Omron CX-Programmer project NuevoProyecto (CX-Programmer 9.31)

# PLC NuevoPLC1: CJ1M CPU11

## Global symbols (name address type ; comment)
C2_FI_CICLE 3101.00 BOOL
C2_MAGATZEM_1_3 3100.00 BOOL
C2_MAGATZEM_2_4 3100.01 BOOL

## Program Cinta2 (cyclic task 0)
Local symbols
AUTO W0.00 BOOL  ; Marca Estat Automatic
BIT_VALIDACIO_SCADA_DESDE_C1 3100.04 BOOL  ; Validació de la emergencia desde el Scada
C2_BE 0.02 BOOL  ; Bolet de Emergència
C2_DM_1_3 0.09 BOOL  ; Detector Magatzem 1-3
C2_DM_2_4 0.11 BOOL  ; Detector Magatzem 2-4
C2_DPC 0.10 BOOL  ; Detector Centre Cinta
C2_EA_0 W130.00 BOOL  ; Etapa Automatic 0
C2_EA_1 W130.01 BOOL  ; Etapa Automatic 1
C2_EA_10 W130.02 BOOL  ; Etapa Automatic 10
C2_EA_11 W130.04 BOOL  ; Etapa Automatic 11
C2_EA_12 W130.05 BOOL  ; Etapa Automatic 12
C2_EA_20 W130.03 BOOL  ; Etapa Automatic 20
C2_EA_21 W130.06 BOOL  ; Etapa Automatic 21
C2_EA_22 W130.07 BOOL  ; Etapa Automatic 22
C2_EA_30 W130.08 BOOL  ; Etapa Automatic 30
C2_EA_31 W130.09 BOOL  ; Etapa Automatic 31
C2_EM_0 W120.00 BOOL  ; Etapa Manual 0
C2_EM_1 W120.01 BOOL  ; Etapa Manual 1
C2_EM_2 W120.02 BOOL  ; Etapa Manual 2
C2_EM_3 W120.03 BOOL  ; Etapa Manual 3
C2_E_A1 W100.00 BOOL
C2_E_A2 W100.03 BOOL
C2_E_D1 W100.06 BOOL
C2_E_D2 W100.07 BOOL
C2_E_F1 W100.01 BOOL
C2_E_F4 W100.04 BOOL
C2_E_F41 W100.05 BOOL
C2_HEMER 1.07 BOOL  ; Pilot Emergència
C2_HMA 1.05 BOOL  ; Pilot mode automàtic
C2_HMM 1.06 BOOL  ; Pilot mode manual
C2_JOYSTICK_FWD 0.03 BOOL  ; Joystick Forward
C2_JOYSTICK_RWD 0.04 BOOL  ; Joystick Reward
C2_MOTOR_FWD 1.09 BOOL  ; Avançament de la cinta
C2_MOTOR_RWD 1.10 BOOL  ; Retrocés de la cinta
C2_PILOT_MARXA 1.00 BOOL  ; Pilot cinta marxa
C2_PM 0.00 BOOL  ; Polsador de Marxa
C2_PP 0.01 BOOL  ; Polsador de Aturada
C2_P_Rearme 0.05 BOOL  ; Polsador de Rearmament
C2_SCADA_JOYSTICK_FWD W101.10 BOOL  ; Joystick SCADA Forward
C2_SCADA_JOYSTICK_RWD W101.11 BOOL  ; Joystick SCADA  Reward
C2_SMA 0.06 BOOL  ; Selector Manual Automatic
CINTA1_REARMADA W300.00 BOOL
COMANDES_SENSE_FINALITZAR 3100.10 BOOL
CT1_MAGATZEM1_3 3100.00 BOOL  ; Ordre peça Magatzem 1-3
CT1_MAGATZEM2_4 3100.01 BOOL  ; Ordre peça Magatzem 2-4
CT2_EMER_LOG 3101.02 BOOL
CT2_FI_CICLE_COM 3101.00 BOOL  ; Ordre de CT2 a CT1, cicle finalitzat
CT2_P_EMER_FIS 3101.03 BOOL
EMER_DESDE_C1 3100.08 BOOL
FI_DE_TOTES_COMADES 3100.09 BOOL
MAN W0.01 BOOL  ; Marca Estat Manual
MEM_FI_COMANDES W100.02 BOOL
M_First_Scan W500.00 BOOL  ; Marca de First Scan
REARMAMENT_C2 W300.10 BOOL
REAR_C1 3100.07 BOOL
REAR_C2 3101.06 BOOL
REAR_CINTES W500.01 BOOL  ; Cinta 1 i Cinta 2 rearmades
RESET_FI_CICLE 3100.05 BOOL
SENYAL_PEÇA_DEIXADA 0.12 BOOL
VAL_TEMPORAL_SCADA W0.08 BOOL

### Section INICIALITZACIÓ_I_ETAPA_ACTIVA_GEMMA

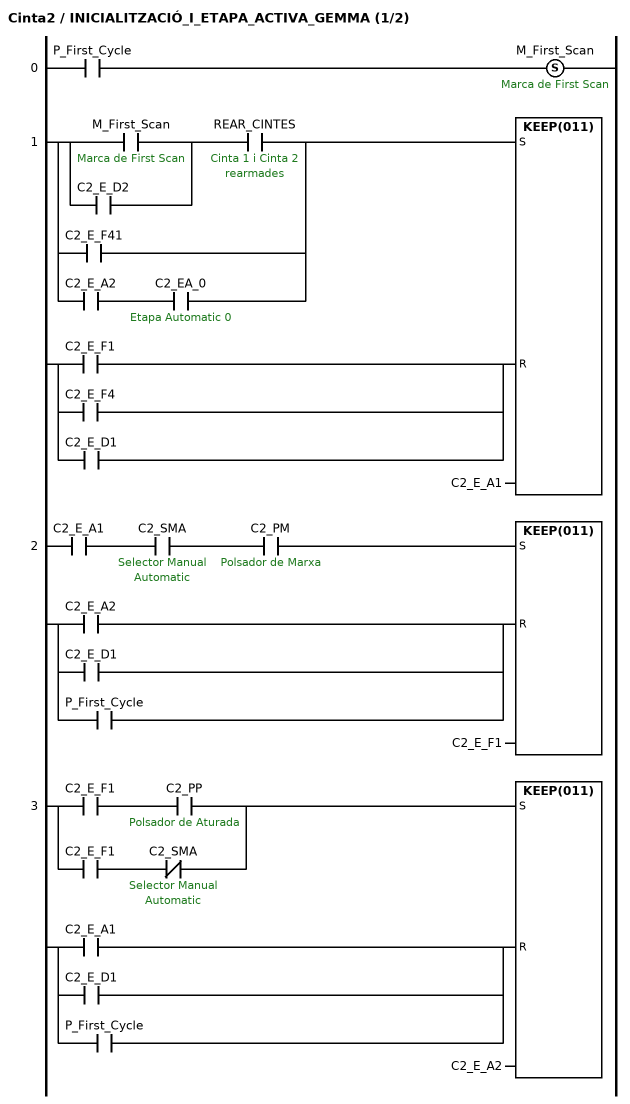
; rung 0
LD P_First_Cycle
SET M_First_Scan  ; Marca de First Scan
; rung 1
LD M_First_Scan  ; Marca de First Scan
OR C2_E_D2
AND REAR_CINTES  ; Cinta 1 i Cinta 2 rearmades
OR C2_E_F41
LD C2_E_A2
AND C2_EA_0  ; Etapa Automatic 0
ORLD
LD C2_E_F1
OR C2_E_F4
OR C2_E_D1
KEEP(011) C2_E_A1
; rung 2
LD C2_E_A1
AND C2_SMA  ; Selector Manual Automatic
AND C2_PM  ; Polsador de Marxa
LD C2_E_A2
OR C2_E_D1
OR P_First_Cycle
KEEP(011) C2_E_F1
; rung 3
LD C2_E_F1
AND C2_PP  ; Polsador de Aturada
LD C2_E_F1
ANDNOT C2_SMA  ; Selector Manual Automatic
ORLD
LD C2_E_A1
OR C2_E_D1
OR P_First_Cycle
KEEP(011) C2_E_A2

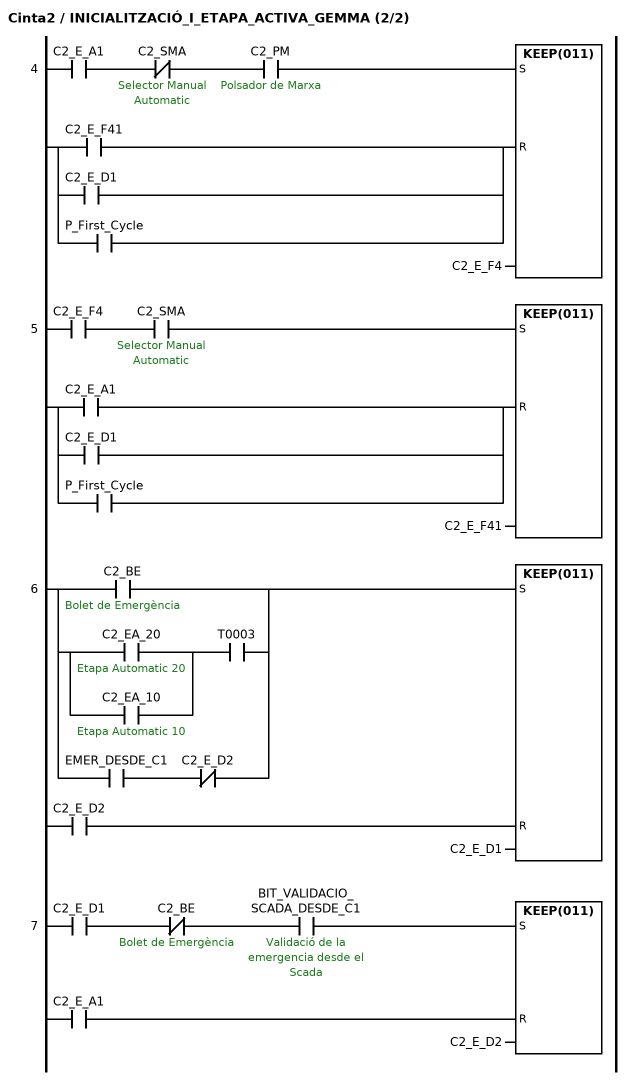
; rung 4
LD C2_E_A1
ANDNOT C2_SMA  ; Selector Manual Automatic
AND C2_PM  ; Polsador de Marxa
LD C2_E_F41
OR C2_E_D1
OR P_First_Cycle
KEEP(011) C2_E_F4
; rung 5
LD C2_E_F4
AND C2_SMA  ; Selector Manual Automatic
LD C2_E_A1
OR C2_E_D1
OR P_First_Cycle
KEEP(011) C2_E_F41
; rung 6
LD C2_BE  ; Bolet de Emergència
LD C2_EA_20  ; Etapa Automatic 20
OR C2_EA_10  ; Etapa Automatic 10
AND T0003
ORLD
LD EMER_DESDE_C1
ANDNOT C2_E_D2
ORLD
LD C2_E_D2
KEEP(011) C2_E_D1
; rung 7
LD C2_E_D1
ANDNOT C2_BE  ; Bolet de Emergència
AND BIT_VALIDACIO_SCADA_DESDE_C1  ; Validació de la emergencia desde el Scada
LD C2_E_A1
KEEP(011) C2_E_D2

### Section ACCIONS_GEMMA

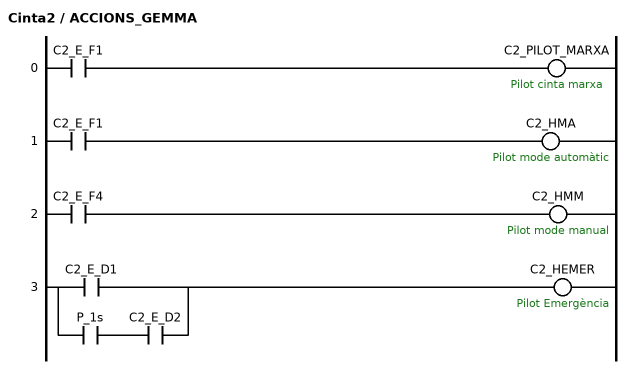
; rung 0
LD C2_E_F1
OUT C2_PILOT_MARXA  ; Pilot cinta marxa
; rung 1
LD C2_E_F1
OUT C2_HMA  ; Pilot mode automàtic
; rung 2
LD C2_E_F4
OUT C2_HMM  ; Pilot mode manual
; rung 3
LD C2_E_D1
LD P_1s
AND C2_E_D2
ORLD
OUT C2_HEMER  ; Pilot Emergència

### Section E_F1

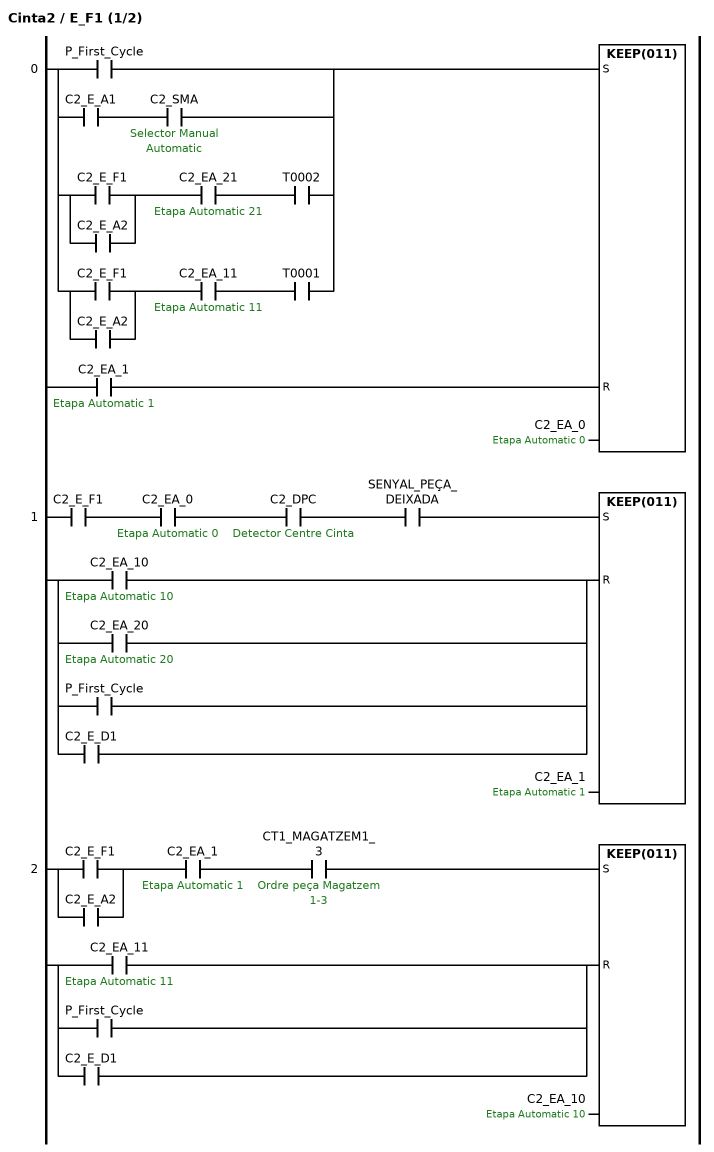
; rung 0
LD P_First_Cycle
LD C2_E_A1
AND C2_SMA  ; Selector Manual Automatic
ORLD
LD C2_E_F1
OR C2_E_A2
AND C2_EA_21  ; Etapa Automatic 21
AND T0002
ORLD
LD C2_E_F1
OR C2_E_A2
AND C2_EA_11  ; Etapa Automatic 11
AND T0001
ORLD
LD C2_EA_1  ; Etapa Automatic 1
KEEP(011) C2_EA_0  ; Etapa Automatic 0
; rung 1
LD C2_E_F1
AND C2_EA_0  ; Etapa Automatic 0
AND C2_DPC  ; Detector Centre Cinta
AND SENYAL_PEÇA_DEIXADA
LD C2_EA_10  ; Etapa Automatic 10
OR C2_EA_20  ; Etapa Automatic 20
OR P_First_Cycle
OR C2_E_D1
KEEP(011) C2_EA_1  ; Etapa Automatic 1
; rung 2
LD C2_E_F1
OR C2_E_A2
AND C2_EA_1  ; Etapa Automatic 1
AND CT1_MAGATZEM1_3  ; Ordre peça Magatzem 1-3
LD C2_EA_11  ; Etapa Automatic 11
OR P_First_Cycle
OR C2_E_D1
KEEP(011) C2_EA_10  ; Etapa Automatic 10

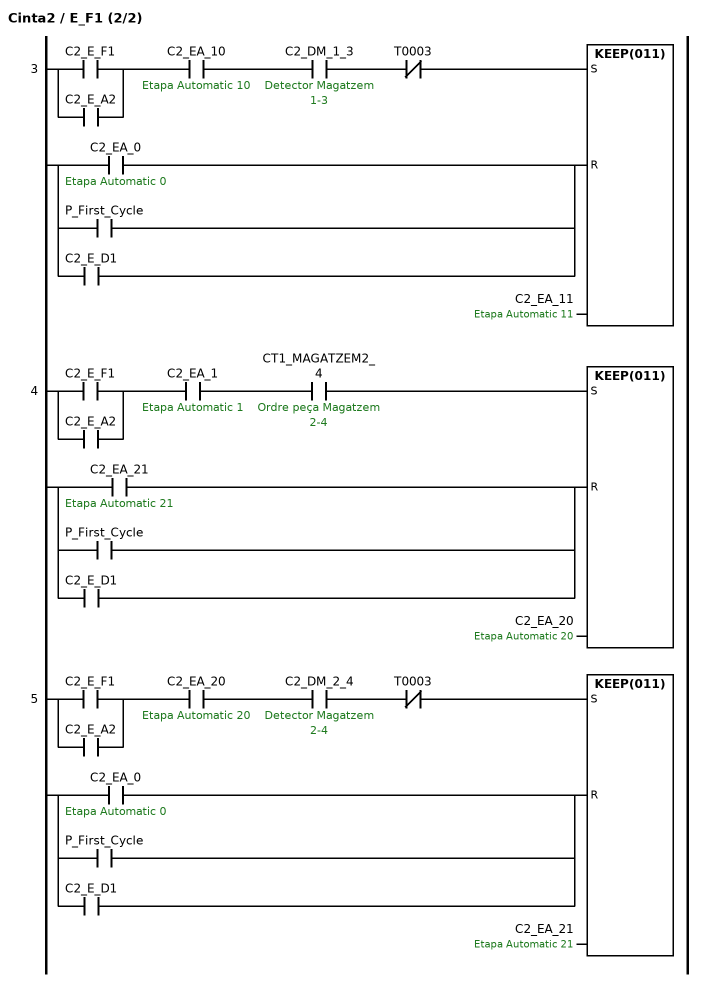
; rung 3
LD C2_E_F1
OR C2_E_A2
AND C2_EA_10  ; Etapa Automatic 10
AND C2_DM_1_3  ; Detector Magatzem 1-3
ANDNOT T0003
LD C2_EA_0  ; Etapa Automatic 0
OR P_First_Cycle
OR C2_E_D1
KEEP(011) C2_EA_11  ; Etapa Automatic 11
; rung 4
LD C2_E_F1
OR C2_E_A2
AND C2_EA_1  ; Etapa Automatic 1
AND CT1_MAGATZEM2_4  ; Ordre peça Magatzem 2-4
LD C2_EA_21  ; Etapa Automatic 21
OR P_First_Cycle
OR C2_E_D1
KEEP(011) C2_EA_20  ; Etapa Automatic 20
; rung 5
LD C2_E_F1
OR C2_E_A2
AND C2_EA_20  ; Etapa Automatic 20
AND C2_DM_2_4  ; Detector Magatzem 2-4
ANDNOT T0003
LD C2_EA_0  ; Etapa Automatic 0
OR P_First_Cycle
OR C2_E_D1
KEEP(011) C2_EA_21  ; Etapa Automatic 21

### Section E_F4

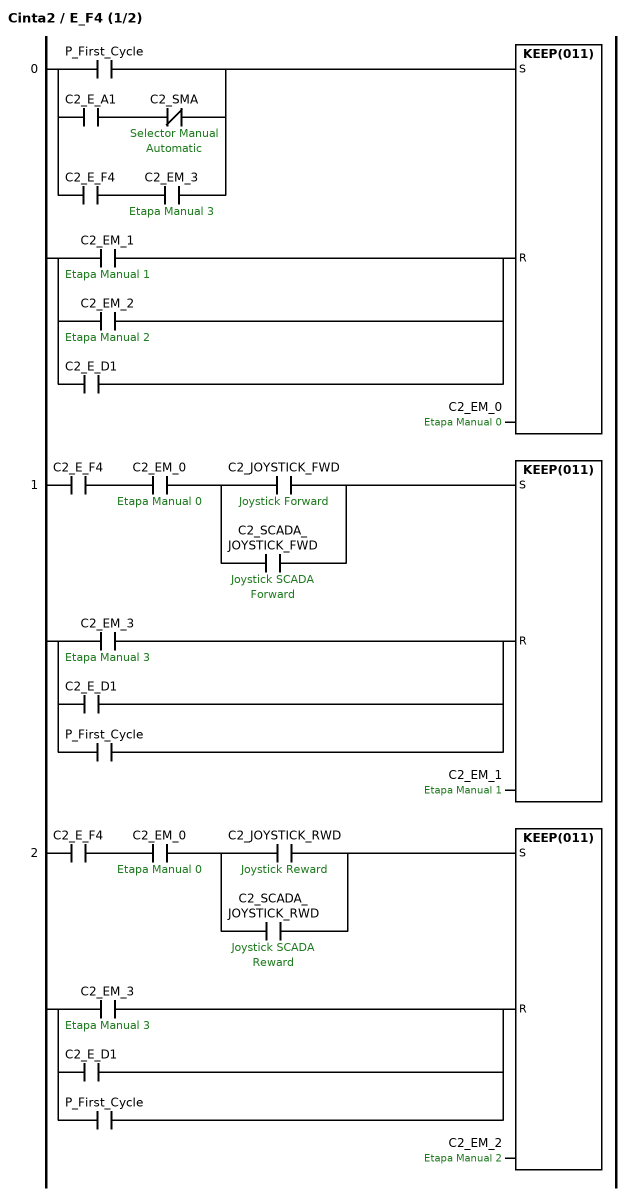
; rung 0
LD P_First_Cycle
LD C2_E_A1
ANDNOT C2_SMA  ; Selector Manual Automatic
ORLD
LD C2_E_F4
AND C2_EM_3  ; Etapa Manual 3
ORLD
LD C2_EM_1  ; Etapa Manual 1
OR C2_EM_2  ; Etapa Manual 2
OR C2_E_D1
KEEP(011) C2_EM_0  ; Etapa Manual 0
; rung 1
LD C2_E_F4
AND C2_EM_0  ; Etapa Manual 0
LD C2_JOYSTICK_FWD  ; Joystick Forward
OR C2_SCADA_JOYSTICK_FWD  ; Joystick SCADA Forward
ANDLD
LD C2_EM_3  ; Etapa Manual 3
OR C2_E_D1
OR P_First_Cycle
KEEP(011) C2_EM_1  ; Etapa Manual 1
; rung 2
LD C2_E_F4
AND C2_EM_0  ; Etapa Manual 0
LD C2_JOYSTICK_RWD  ; Joystick Reward
OR C2_SCADA_JOYSTICK_RWD  ; Joystick SCADA  Reward
ANDLD
LD C2_EM_3  ; Etapa Manual 3
OR C2_E_D1
OR P_First_Cycle
KEEP(011) C2_EM_2  ; Etapa Manual 2

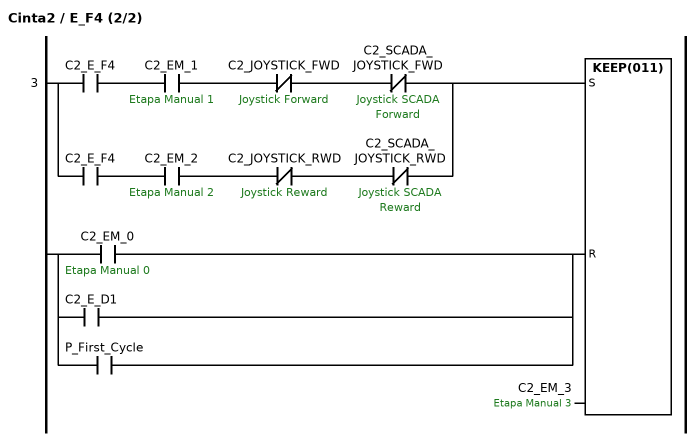
; rung 3
LD C2_E_F4
AND C2_EM_1  ; Etapa Manual 1
ANDNOT C2_JOYSTICK_FWD  ; Joystick Forward
ANDNOT C2_SCADA_JOYSTICK_FWD  ; Joystick SCADA Forward
LD C2_E_F4
AND C2_EM_2  ; Etapa Manual 2
ANDNOT C2_JOYSTICK_RWD  ; Joystick Reward
ANDNOT C2_SCADA_JOYSTICK_RWD  ; Joystick SCADA  Reward
ORLD
LD C2_EM_0  ; Etapa Manual 0
OR C2_E_D1
OR P_First_Cycle
KEEP(011) C2_EM_3  ; Etapa Manual 3

### Section ACCIONS

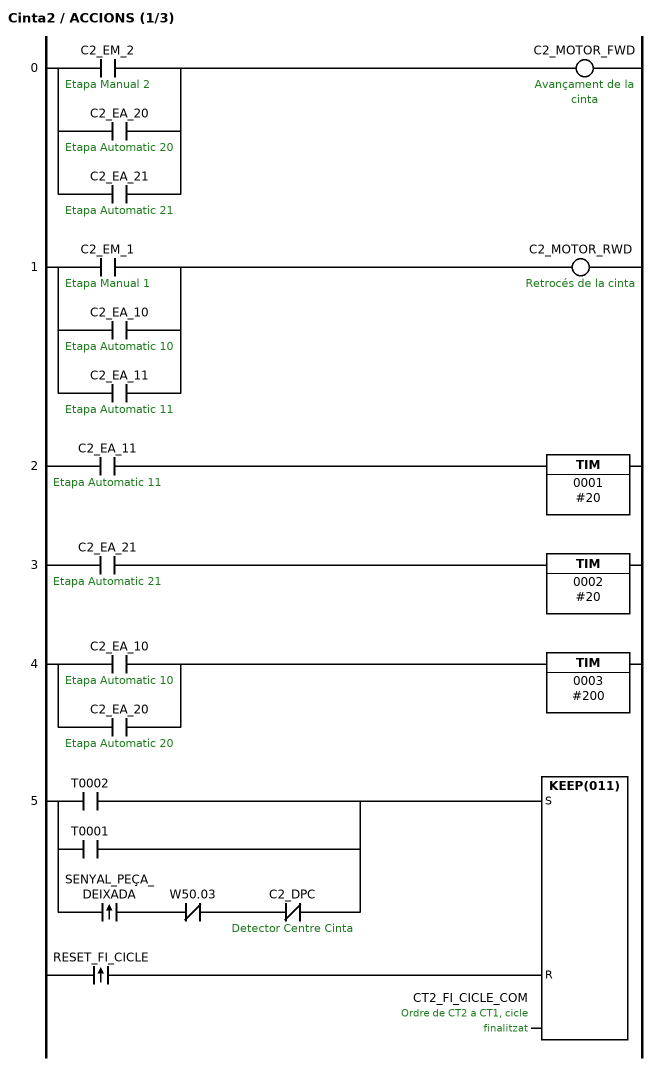
; rung 0
LD C2_EM_2  ; Etapa Manual 2
OR C2_EA_20  ; Etapa Automatic 20
OR C2_EA_21  ; Etapa Automatic 21
OUT C2_MOTOR_FWD  ; Avançament de la cinta
; rung 1
LD C2_EM_1  ; Etapa Manual 1
OR C2_EA_10  ; Etapa Automatic 10
OR C2_EA_11  ; Etapa Automatic 11
OUT C2_MOTOR_RWD  ; Retrocés de la cinta
; rung 2
LD C2_EA_11  ; Etapa Automatic 11
TIM 0001 #20
; rung 3
LD C2_EA_21  ; Etapa Automatic 21
TIM 0002 #20
; rung 4
LD C2_EA_10  ; Etapa Automatic 10
OR C2_EA_20  ; Etapa Automatic 20
TIM 0003 #200
; rung 5
LD T0002
OR T0001
@LD SENYAL_PEÇA_DEIXADA
ANDNOT W50.03
ANDNOT C2_DPC  ; Detector Centre Cinta
ORLD
@LD RESET_FI_CICLE
KEEP(011) CT2_FI_CICLE_COM  ; Ordre de CT2 a CT1, cicle finalitzat

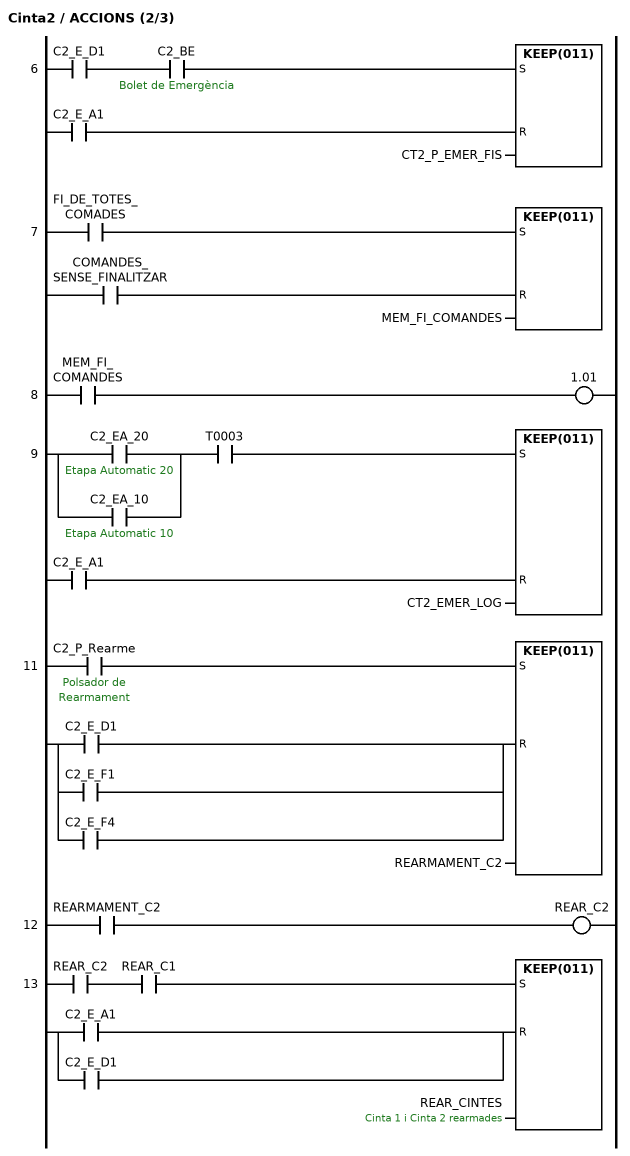
; rung 6
LD C2_E_D1
AND C2_BE  ; Bolet de Emergència
LD C2_E_A1
KEEP(011) CT2_P_EMER_FIS
; rung 7
LD FI_DE_TOTES_COMADES
LD COMANDES_SENSE_FINALITZAR
KEEP(011) MEM_FI_COMANDES
; rung 8
LD MEM_FI_COMANDES
OUT 1.01
; rung 9
LD C2_EA_20  ; Etapa Automatic 20
OR C2_EA_10  ; Etapa Automatic 10
AND T0003
LD C2_E_A1
KEEP(011) CT2_EMER_LOG
; rung 11
LD C2_P_Rearme  ; Polsador de Rearmament
LD C2_E_D1
OR C2_E_F1
OR C2_E_F4
KEEP(011) REARMAMENT_C2
; rung 12
LD REARMAMENT_C2
OUT REAR_C2
; rung 13
LD REAR_C2
AND REAR_C1
LD C2_E_A1
OR C2_E_D1
KEEP(011) REAR_CINTES  ; Cinta 1 i Cinta 2 rearmades

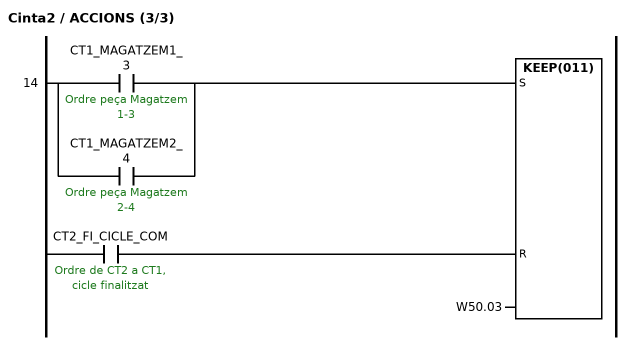
; rung 14
LD CT1_MAGATZEM1_3  ; Ordre peça Magatzem 1-3
OR CT1_MAGATZEM2_4  ; Ordre peça Magatzem 2-4
LD CT2_FI_CICLE_COM  ; Ordre de CT2 a CT1, cicle finalitzat
KEEP(011) W50.03

### Section ACCIONS_HMI

### Section END
; rung 0
END(001)